(* CoDeSys 2.3 export: CHARCODE.EXP *)

(* POU 05_Basic_Calc/CHARCODE, ST *)
FUNCTION CHARCODE : BYTE
(* Функция получает код (char) для текстового символа *)
VAR_INPUT
	STR : STRING(1);
END_VAR
VAR
	PT : POINTER TO BYTE;
END_VAR
PT := ADR(STR);
CHARCODE := PT^;
END_FUNCTION
